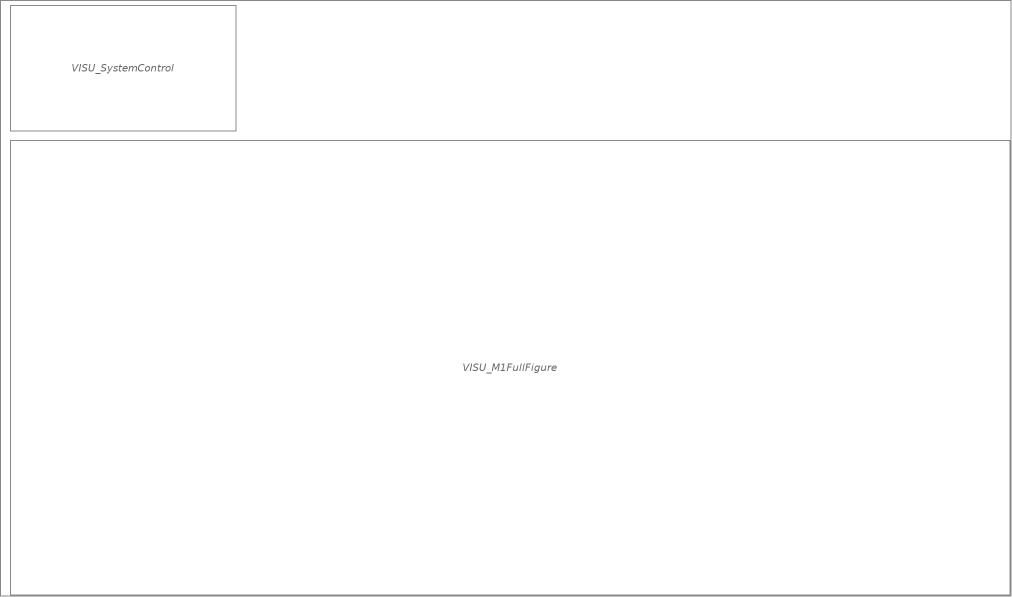
VISUALIZATION VISU_M1Overview  // 1012x597
VAR_IN_OUT
	ref : M1;
    widget : M1Widget;
END_VAR
    Frame (10,5 226x126)
        shows VISU_SystemControl(status := widget.actualStatus, button_initialize := widget.button_initialize, button_operating := widget.button_operating, button_locking := widget.button_locking)
    Frame (10,140 1000x455)
        shows VISU_M1FullFigure(ref := ref, widget := widget)
END_VISUALIZATION

(* stored: Version 1.1.0.1, ProductVersion 3.1.4019.2
   Visu VISU_M1Overview: Id {990d383a-b93a-4984-b387-5e3b9b3bc924} *)
